(* Logix 5000 project; controller Test_Bench vendor 1 type 14 code 155 rev 34.11; software revision 34.00; part 2 of 2 *)

ADD_ON_INSTRUCTION Analog_Scale   (* revision 1.0, vendor Jeya Prakash *)
VAR_INPUT
   Analog_In : REAL; {required}   // unscaled analog input
   Analog_Min_In : REAL; {required}   // MINIMUM ENGINEERING UNITS TO SCALE
   Analog_Max_In : REAL; {required}   // MAXIMUM ENGINEERING UNITS TO SCALE
   Low_Clamp_Value : REAL; {required}   // USED TO CALCULATE THE RANGE OF THE SCALING
   High_Clamp_Value : REAL; {required}   // USED TO CALCULATE THE RANGE OF THE SCALING
END_VAR
VAR_OUTPUT
   Analog_Out : REAL; {access Read Only, required}   // THE RESULT OF THE CALCULATION IN UNITS THAT WORK WITH THE COMPACTLOGIX ANALOG MODULE WITH THE OFFSET FROM ZERO ADDED IN
END_VAR

ROUTINE Logic   (* ladder *)
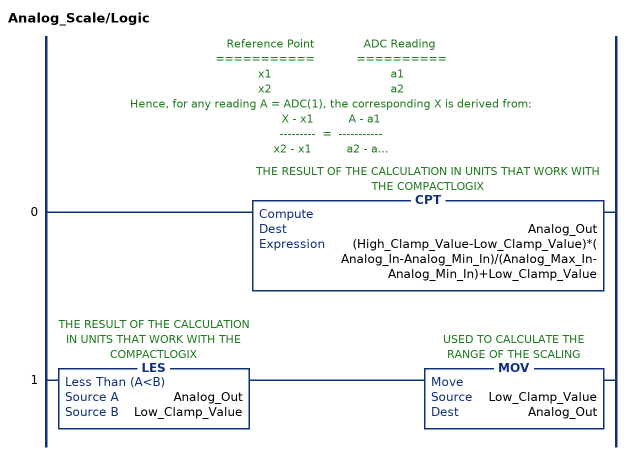
   // Reference Point              ADC Reading
   // ===========            ==========
   //       x1                                  a1
   //       x2                                  a2
   // Hence, for any reading A = ADC(1), the corresponding X is derived from:
   //   X - x1          A - a1
   // ---------  =  -----------
   // x2 - x1          a2 - a1
   // ==>  X = (x2 - x1)*(A - a1)/(a2 - a1) + x1
   // Note that since x1,x2,a1, and a2 are all constants the actual formula is much simpler then it appears above.
   // E.g. Temperature measurement
   // ========================
   //     Temp            ADC(n)
   //         30              200
   //       100              3000
   // So for any ADC readings A, the temperature is:
   //   X = 70*(A - 200)/2800 + 30
   // Note: To get better resolution , you can represent 30 degree as 300 and 100 degree as 1000 so if X = 123 it means 12.3 degree.
   0: CPT(Analog_Out,(High_Clamp_Value-Low_Clamp_Value)*(Analog_In-Analog_Min_In)/(Analog_Max_In-Analog_Min_In)+Low_Clamp_Value);
   1: LES(Analog_Out,Low_Clamp_Value)MOV(Low_Clamp_Value,Analog_Out);
END_ROUTINE
END_ADD_ON_INSTRUCTION

ADD_ON_INSTRUCTION Generic_8PORT_IOL   (* revision 3.0 *)
// Revision note:
// 12/2022:updated to current AOI standards:LH
VAR_IN_OUT
   PLC_Input : INT[223]; {required}   // Reference the Input Controller tag <IOLinkMasterName>:I1.Data
   PLC_Output : INT[151]; {required}   // Reference the Output Controller tag <IOLinkMasterName>:O1.Data
END_VAR
VAR_INPUT
   Port_Process_Data_Size : SINT := 4;   // User Input Value from the Configuration Controller tag <IOLinkMasterName>:C.Port_Process_Data_Size
   Port_Number : SINT; {visible}   // User Input Value = Port number of the IO-Link Master
END_VAR
VAR_OUTPUT
   Vendor_ID : INT; {access Read Only, visible}   // Read only value indicating the manufacturer of the IO-Link Device. ifm=310 dec
   Device_ID : DINT; {access Read Only, visible}   // Read only value set by the manufacturer of the device. Varies by product family
   IOL_Mode : BOOL; {access Read Only, visible}   // True: Port is configured for IO-Link Communication. False: Port is not configured for IO-Link Communication
   Device_Not_Connected : BOOL; {access Read Only, visible}   // True: No IO-Link Device is connected False: IO-Link Device is connected
   Invalid_Data : BOOL; {access Read Only, visible}   // True: IO-Link Data is invalid False: IO-Link Data is valid
   Wrong_VID_DID : BOOL; {access Read Only, visible}   // True: Vendor ID and/or Device ID does not match the configured VID or DID set in Configuration Controller Tag(s) <IOLink MasterName>:C.Vendor_ID_Port_n or ...C.Device_ID_Port_n
   Diagnostic_Avail : BOOL; {access Read Only, visible}   // True: IO-Link Event data is available False: No Event data is present
   AOI_Settings_Error : BOOL; {access Read Only, visible}   // A user input is out of range. Check port process data size and port number
END_VAR
VAR_IN_OUT
   Input_Data_Array : INT[16]; {required}   // Up to 16 words/32 bytes of Input process data produced by the IO-Link device
        [0]   // Input Word 0/Byte 0 0..7/Byte 1 8..15
        [1]   // Input Word 1/Byte 2 0..7/Byte 3 8..15
        [10]   // Input Word 10/Byte 20 0..7/Byte 21 8..15
        [11]   // Input Word 11/Byte 22 0..7/Byte 23 8..15
        [12]   // Input Word 12/Byte 24 0..7/Byte 25 8..15
        [13]   // Input Word 13/Byte 26 0..7/Byte 27 8..15
        [14]   // Input Word 14/Byte 28 0..7/Byte 29 8..15
        [15]   // Input Word 15/Byte 30 0..7/Byte 31 8..15
        [2]   // Input Word 2/Byte 4 0..7/Byte 5 8..15
        [3]   // Input Word 3/Byte 6 0..7/Byte 7 8..15
        [4]   // Input Word 4/Byte 8 0..7/Byte 9 8..15
        [5]   // Input Word 5/Byte 10 0..7/Byte 11 8..15
        [6]   // Input Word 6/Byte 12 0..7/Byte 13 8..15
        [7]   // Input Word 7/Byte 14 0..7/Byte 15 8..15
        [8]   // Input Word 8/Byte 16 0..7/Byte 17 8..15
        [9]   // Input Word 9/Byte 18 0..7/Byte 19 8..15
   Output_Data_Array : INT[16]; {required}   // Up to 32 bytes of Output process data consumed by the IO-Link device
        [7]   // Output Word 7/Byte 15 0..7/Byte 14 8..15
        [8]   // Output Word 8/Byte 17 0..7/Byte 16 8..15
        [9]   // Output Word 9/Byte 19 0..7/Byte 18 8..15
        [0]   // Output Word 0/Byte 1 0..7/Byte 0 8..15
        [10]   // Output Word 10/Byte 21 0..7/Byte 20 8..15
        [11]   // Output Word 11/Byte 23 0..7/Byte 22 8..15
        [12]   // Output Word 12/Byte 25 0..7/Byte 24 8..15
        [13]   // Output Word 13/Byte 27 0..7/Byte 26 8..15
        [14]   // Output Word 14/Byte 29 0..7/Byte 28 8..15
        [15]   // Output Word 15/Byte 31 0..7/Byte 30 8..15
        [1]   // Output Word 1/Byte 3 0..7/Byte 2 8..15
        [2]   // Output Word 2/Byte 5 0..7/Byte 4 8..15
        [3]   // Output Word 3/Byte 7 0..7/Byte 6 8..15
        [4]   // Output Word 4/Byte 9 0..7/Byte 8 8..15
        [5]   // Output Word 5/Byte 11 0..7/Byte 10 8..15
        [6]   // Output Word 6/Byte 13 0..7/Byte 12 8..15
END_VAR
VAR
   Data_Size : SINT; {access None}   // Factor of the RealPort_Num to calcualated the Offset_Address
   Offset_StatusFlgs : SINT; {access None}   // RealPort_Num+9
   RealPort_Num : SINT; {access None}   // Result of the Port_Number-1
   StatusFlgs_Offset : SINT; {access None}   // Result of Offset_StatusFlgs+23
   Offset_Address : INT; {access None}   // Result of Data_Size*RealPort_Number
   Process_Offset : INT; {access None}   // Result of Offset_Address+95(8port Master) or Offset_Address+59(4port Master). Used to indicate the word offset for where the IO-Link device’s process input data starts
   Process_Out_Offset : INT; {access None}   // Result of Offset_Address+23
END_VAR

ROUTINE Logic   (* ladder *)
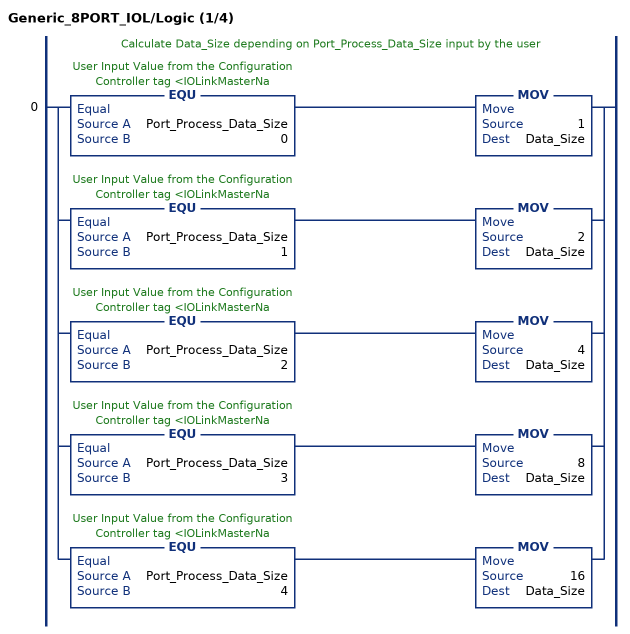
   // Calculate Data_Size depending on Port_Process_Data_Size input by the user
   0: [EQU(Port_Process_Data_Size,0) MOV(1,Data_Size) ,EQU(Port_Process_Data_Size,1) MOV(2,Data_Size) ,EQU(Port_Process_Data_Size,2) MOV(4,Data_Size) ,EQU(Port_Process_Data_Size,3) MOV(8,Data_Size) ,EQU(Port_Process_Data_Size,4) MOV(16,Data_Size) ];
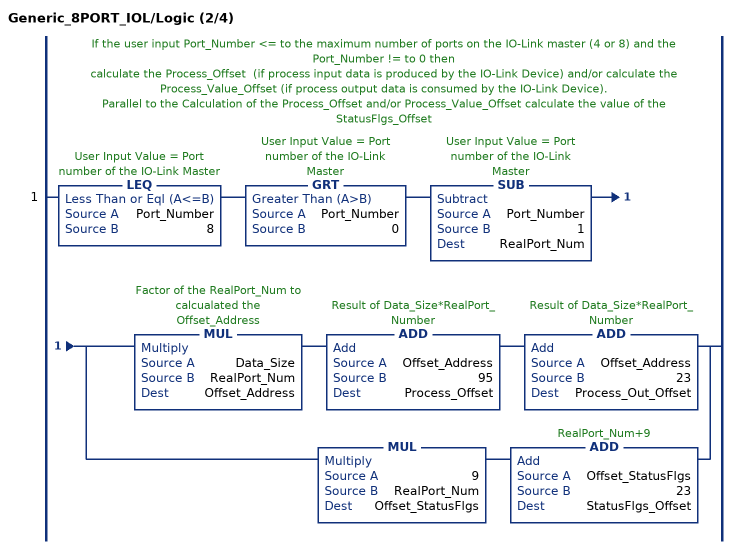
   // If the user input Port_Number <= to the maximum number of ports on the IO-Link master (4 or 8) and the Port_Number != to 0 then
   // calculate the Process_Offset  (if process input data is produced by the IO-Link Device) and/or calculate the Process_Value_Offset (if process output data is consumed by the IO-Link Device).
   // Parallel to the Calculation of the Process_Offset and/or Process_Value_Offset calculate the value of the StatusFlgs_Offset
   1: LEQ(Port_Number,8)GRT(Port_Number,0)SUB(Port_Number,1,RealPort_Num)[MUL(Data_Size,RealPort_Num,Offset_Address) ADD(Offset_Address,95,Process_Offset) ADD(Offset_Address,23,Process_Out_Offset) ,MUL(9,RealPort_Num,Offset_StatusFlgs) ADD(Offset_StatusFlgs,23,StatusFlgs_Offset) ];
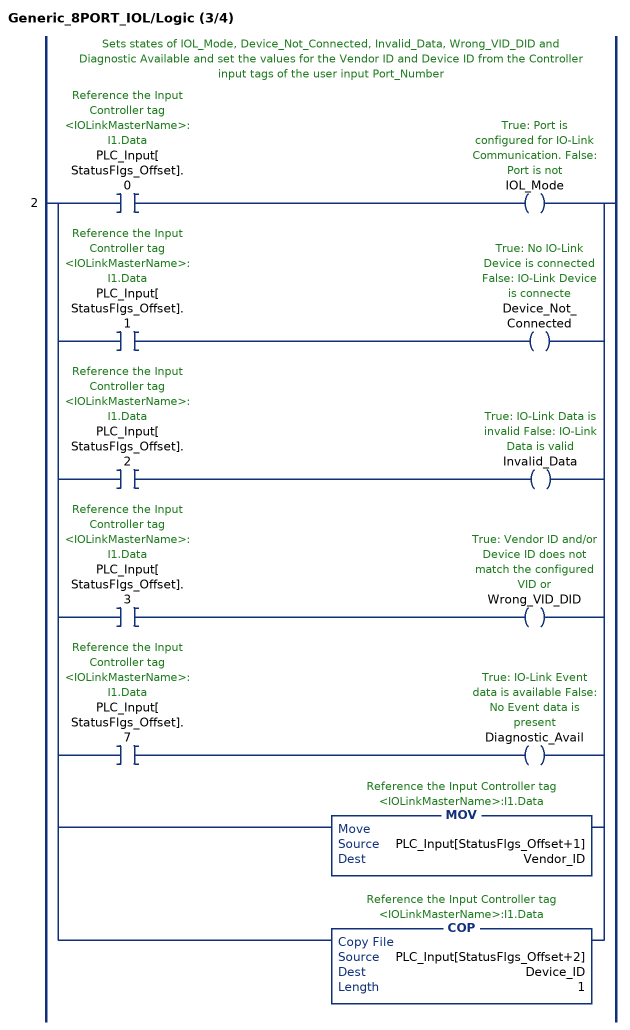
   // Sets states of IOL_Mode, Device_Not_Connected, Invalid_Data, Wrong_VID_DID and Diagnostic Available and set the values for the Vendor ID and Device ID from the Controller input tags of the user input Port_Number
   2: [XIC(PLC_Input[StatusFlgs_Offset].0) OTE(IOL_Mode) ,XIC(PLC_Input[StatusFlgs_Offset].1) OTE(Device_Not_Connected) ,XIC(PLC_Input[StatusFlgs_Offset].2) OTE(Invalid_Data) ,XIC(PLC_Input[StatusFlgs_Offset].3) OTE(Wrong_VID_DID) ,XIC(PLC_Input[StatusFlgs_Offset].7) OTE(Diagnostic_Avail) ,MOV(PLC_Input[StatusFlgs_Offset+1],Vendor_ID) ,COP(PLC_Input[StatusFlgs_Offset+2],Device_ID,1) ];
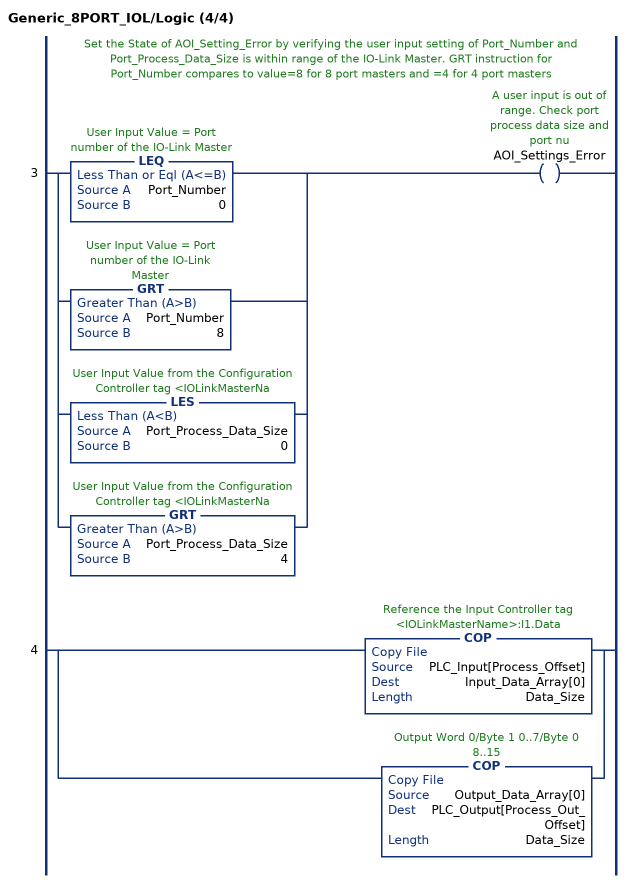
   // Set the State of AOI_Setting_Error by verifying the user input setting of Port_Number and Port_Process_Data_Size is within range of the IO-Link Master. GRT instruction for Port_Number compares to value=8 for 8 port masters and =4 for 4 port masters
   3: [LEQ(Port_Number,0) ,GRT(Port_Number,8) ,LES(Port_Process_Data_Size,0) ,GRT(Port_Process_Data_Size,4) ]OTE(AOI_Settings_Error);
   4: [COP(PLC_Input[Process_Offset],Input_Data_Array[0],Data_Size) ,COP(Output_Data_Array[0],PLC_Output[Process_Out_Offset],Data_Size) ];
END_ROUTINE
END_ADD_ON_INSTRUCTION

ADD_ON_INSTRUCTION Hour_Meter   (* revision 1.0 *)
// Counts Run hours
VAR_OUTPUT
   output_hours : DINT := 250; {access Read Only, required}
END_VAR
VAR
   timers : TIMER[3] := ([0].PRE := 3600000, [0].ACC := 2154); {access None}
   Internal_Hours : COUNTER := (ACC := 1131); {access None}
   start_timer : DINT; {access None}
END_VAR

ROUTINE Logic   (* ladder *)
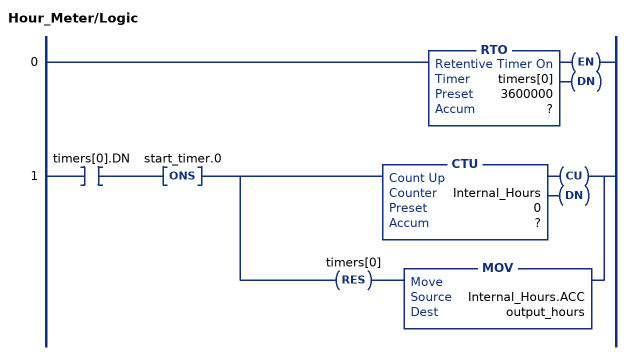
   0: RTO(timers[0],?,?);
   1: XIC(timers[0].DN)ONS(start_timer.0)[CTU(Internal_Hours,?,?) ,RES(timers[0]) MOV(Internal_Hours.ACC,output_hours) ];
END_ROUTINE
END_ADD_ON_INSTRUCTION

VAR_GLOBAL   (* controller tags *)
   AOI_hours : DINT := 14;
   AOI_timer : DINT;
   Axis_Init_State : DINT;
   BOOL : BOOL[64] := ([3] := 1);
        [3]   // Run Meter Enable
        [4]   // Enable Motion Gear
   Comms : DINT;
   ConfigBuff : INT[5];
   ConfigBuffer : DINT;
   Counters : COUNTER[20] := ([0].ACC := 1624, [0].DN := 1);
        [0]   // Hour Meter
   enc : AXIS_CIP_DRIVE;
   Message : MESSAGE;
        MessageParameters(ServiceCode := 16#0fa2, LocalElement := SLC_Read[0], ...)
   motion_control : MOTION_INSTRUCTION[16];
   servo_drive : AXIS_CIP_DRIVE;
   SLC_Read : INT[1] := ([0] := -14432);
   Temp : DINT := 51;
   temp3 : Analog_Scale := (Analog_In := 6058.0, Analog_Min_In := 4000.0, Analog_Max_In := 20000.0, Low_Clamp_Value := 14.0, High_Clamp_Value := 302.0, Analog_Out := 51.044);
   test : MOTION_GROUP;
   Time : DINT[7] := ([0] := 2023, [1] := 1, [2] := 27, [3] := 18, [4] := 57, [5] := 41, [6] := 913003);
   Timers : TIMER[20] := ([0].PRE := 2000, [0].ACC := 1647, [0].EN := 1, [0].TT := 1);
        [0]   // SecondsToHours
END_VAR

PROGRAM MainProgram   (* main routine MainRoutine *)
VAR
   DFF_01 : FLIP_FLOP_D;
   InputData : INT[16];
   IOLINK : DINT;
   OutputData : INT[16];
   Sensor : Generic_8PORT_IOL := (Port_Process_Data_Size := 4, Port_Number := 2);
END_VAR

ROUTINE MainRoutine   (* ladder *)
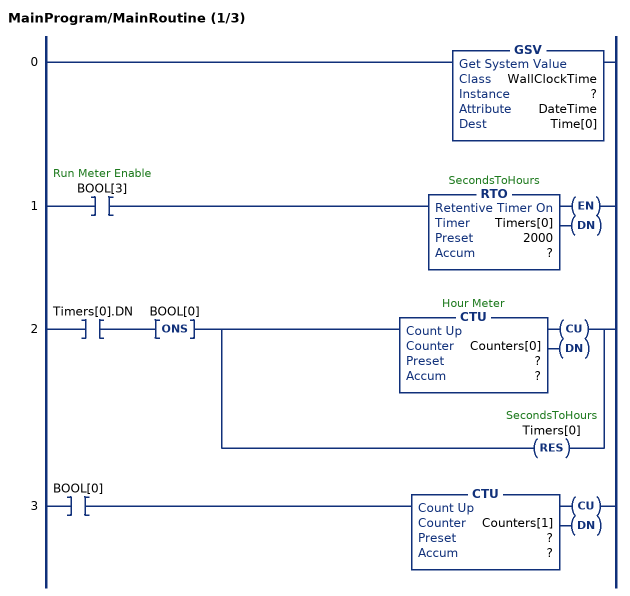
   0: GSV(WallClockTime,?,DateTime,Time[0]);
   1: XIC(BOOL[3])RTO(Timers[0],?,?);
   2: XIC(Timers[0].DN)ONS(BOOL[0])[CTU(Counters[0],?,?) ,RES(Timers[0]) ];
   3: XIC(BOOL[0])CTU(Counters[1],?,?);
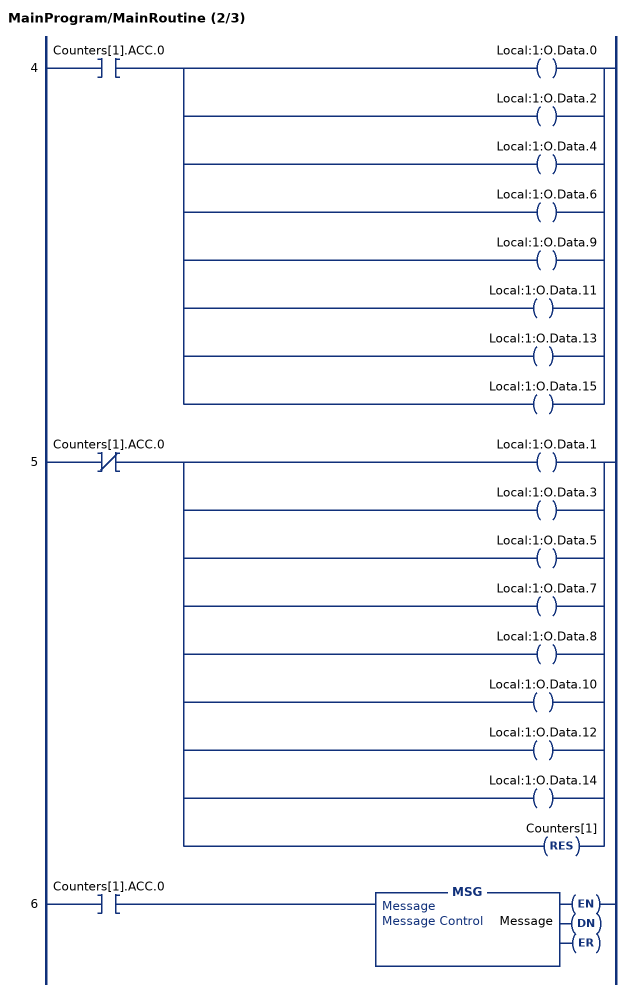
   4: XIC(Counters[1].ACC.0)[OTE(Local:1:O.Data.0) ,OTE(Local:1:O.Data.2) ,OTE(Local:1:O.Data.4) ,OTE(Local:1:O.Data.6) ,OTE(Local:1:O.Data.9) ,OTE(Local:1:O.Data.11) ,OTE(Local:1:O.Data.13) ,OTE(Local:1:O.Data.15) ];
   5: XIO(Counters[1].ACC.0)[OTE(Local:1:O.Data.1) ,OTE(Local:1:O.Data.3) ,OTE(Local:1:O.Data.5) ,OTE(Local:1:O.Data.7) ,OTE(Local:1:O.Data.8) ,OTE(Local:1:O.Data.10) ,OTE(Local:1:O.Data.12) ,OTE(Local:1:O.Data.14) ,RES(Counters[1]) ];
   6: XIC(Counters[1].ACC.0)MSG(Message);
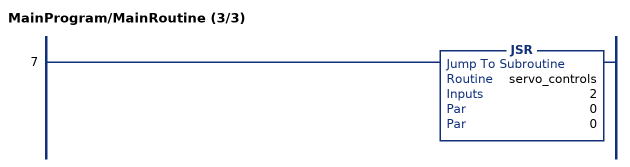
   7: JSR(servo_controls,2,0,0);
END_ROUTINE

ROUTINE servo_controls   (* ladder *)
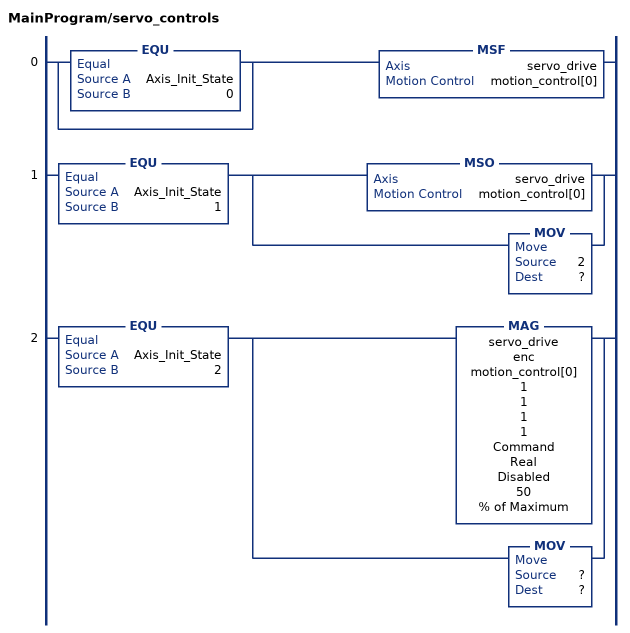
   0: [EQU(Axis_Init_State,0) ,]MSF(servo_drive,motion_control[0]);
   1: EQU(Axis_Init_State,1)[MSO(servo_drive,motion_control[0]) ,MOV(2,?) ];
   2: EQU(Axis_Init_State,2)[MAG(servo_drive,enc,motion_control[0],1,1,1,1,Command,Real,Disabled,50,% of Maximum) ,MOV(?,?) ];
END_ROUTINE
END_PROGRAM
